(* CODESYS project genmed-LogGenTestSP14.project

Project tree, tasks and I/O mapping:
  Device : CODESYS Control for Raspberry Pi MC SL, 3S - Smart Software Solutions GmbH, version 3.5.14.20
    application Application
      libraries: Standard, * (System); VisuGlobalClientManager, * (System)
      task Task (cyclic, interval t#20ms, priority 1) calls PLC_PRG
      task DataLogHighTask (cyclic, interval t#5ms, priority 1) calls AC_CALL_DataLogHighTask_START, AC_CALL_DataLogHighTask_END
      task DataLogLowTask (cyclic, interval t#20ms, priority 10) calls AC_CALL_DataLogLowTask_START, AC_CALL_DataLogLowTask_END
      task AC_GenVisu_Task (cyclic, interval t#50ms, priority 30) calls AC_GenVisu_Prg
      task VISU_TASK (cyclic, interval 100 ms, priority 31) calls VisuElems.Visu_Prg
      program PLC_PRG [ST]
      AC_Std/
        program AC_CALL_DataLogHighTask_START [ST]
        function AC_Init [ST]
        global variables GVL_MODULE_TREE
        program AC_CALL_DataLogHighTask_END [ST]
        function AC_InitInternal [ST]
        function AC_OnlineChange [ST]
        global variables MODULE_INFOS
        program AC_CALL_DataLogLowTask_START [ST]
        program AC_CALL_DataLogLowTask_END [ST]
        global variables GVL_DataLogManager
      data type LogStruct
      data type LogUnion
      AC_Visu/
        function block AC_Visu_FB [ST]: OnFrameIndexChanged, GetModuleFrameIndex, GetAncestor
        visualisation Page_DataLogManager
        function AC_VisuInit [ST]
        visualisation Toplevel
        global variables GVL_Visu
        program AC_GenVisu_Prg [ST]
        function block AC_GlobalClientManagerListener [ST]: ClientDestroyed, ClientCreated
        global variables GVL_GlobalClientManagerListener
        function AC_RegisterVisuClientInit [ST]
      AC_FBs/
        function block AC_DataLogManager_DataLogChannel_1 [ST]
        function block AC_DataLogManager [ST]
        function block AC_DataLogManager_DataLogChannel_1_DataLogStorage_CSV [ST]
        function block AC_DataLogManager_DataLogChannel [ST]
      function block POU_Log [ST]: Prop_Log
      text DataLogConfig
    SoftMotion General Axis Pool
    I²C
    SPI
    GPIOs_A_B : GPIOs A/B, 3S - Smart Software Solutions GmbH, version 3.5.11.0
        unmapped channels: digital inputs (GPIO0..GPIO31), digital outputs (GPIO0..GPIO31)
    Onewire
    Camera device
      <Empty>
  libraries: AC_ModuleBase, * (3S - Smart Software Solutions GmbH); AC_DataLog, 3.5.14.0 (3S - Smart Software Solutions GmbH); AC_Persistence, * (3S - Smart Software Solutions GmbH); VisuSymbols, 3.5.10.0 (System)
  DataLogManager
    DataLogChannels_Role (DataLogChannels)
      DataLogChannel
        DataLogStorage_SQLite
        DataLogStorage_Role (DataLogStorage)
      DataLogChannel_1
        DataLogStorage_CSV
        A storage module. (DataLogStorage)
  AC_GENERATOR_DATA
  text list GlobalTextList
*)

// Device/Application/LogStruct
TYPE LogStruct :
STRUCT
    bNoLog : BOOL;
    {attribute 'ac_datalog'}
    bLog : BOOL;
END_STRUCT
END_TYPE

// Device/Application/LogUnion
TYPE LogUnion :
UNION
    iLog : INT;
    uiLog : UINT;
    wLog : WORD;
END_UNION
END_TYPE

// Device/Application/AC_Std/GVL_MODULE_TREE
//Code generated by Application Composer.
//Modifying generated code is not recommended!

VAR_GLOBAL
	Module_Tree: AC.ModuleTree;
	aNodes: ARRAY[0..5] OF AC.MNode;
	AC_Environment: AC.MEnv;
END_VAR

// Device/Application/AC_Std/MODULE_INFOS
//Code generated by Application Composer.
//Modifying generated code is not recommended!
{attribute 'global_init_slot' := '40000'}
{attribute 'init_on_onlchange'}

VAR_GLOBAL
	{attribute 'init_on_onlchange'}
	AC_DataLog_DataLogManager_INFO: AC.ModuleInfo := (pbyModuleType := ADR('AC_DataLog.DataLogManager'));
	{attribute 'init_on_onlchange'}
	AC_DataLog_DataLogChannel_INFO: AC.ModuleInfo := (pbyModuleType := ADR('AC_DataLog.DataLogChannel'));
	{attribute 'init_on_onlchange'}
	AC_DataLog_DataLogStorage_SQLite_INFO: AC.ModuleInfo := (pbyModuleType := ADR('AC_DataLog.DataLogStorage_SQLite'));
	{attribute 'init_on_onlchange'}
	AC_DataLog_DataLogStorage_CSV_INFO: AC.ModuleInfo := (pbyModuleType := ADR('AC_DataLog.DataLogStorage_CSV'));
END_VAR

// Device/Application/AC_Visu/GVL_Visu
//Code generated by Application Composer.
//Modifying generated code is not recommended!

VAR_GLOBAL
	g_aACVisu: ARRAY[0..7] OF AC_Visu_FB;
	AC_Visu_Dummy: AC_Visu_FB;
	g_aACVisuPtr: ARRAY[-1..127] OF POINTER TO AC_Visu_FB := [ADR(AC_Visu_Dummy), ADR(g_aACVisu[0]), ADR(g_aACVisu[1]), ADR(g_aACVisu[2]), ADR(g_aACVisu[3]), ADR(g_aACVisu[4]), ADR(g_aACVisu[5]), ADR(g_aACVisu[6]), ADR(g_aACVisu[7]), ADR(AC_Visu_Dummy), ADR(AC_Visu_Dummy), ADR(AC_Visu_Dummy), ADR(AC_Visu_Dummy), ADR(AC_Visu_Dummy), ADR(AC_Visu_Dummy), ADR(AC_Visu_Dummy), ADR(AC_Visu_Dummy), ADR(AC_Visu_Dummy), ADR(AC_Visu_Dummy), ADR(AC_Visu_Dummy), ADR(AC_Visu_Dummy), ADR(AC_Visu_Dummy), ADR(AC_Visu_Dummy), ADR(AC_Visu_Dummy), ADR(AC_Visu_Dummy), ADR(AC_Visu_Dummy), ADR(AC_Visu_Dummy), ADR(AC_Visu_Dummy), ADR(AC_Visu_Dummy), ADR(AC_Visu_Dummy), ADR(AC_Visu_Dummy), ADR(AC_Visu_Dummy), ADR(AC_Visu_Dummy), ADR(AC_Visu_Dummy), ADR(AC_Visu_Dummy), ADR(AC_Visu_Dummy), ADR(AC_Visu_Dummy), ADR(AC_Visu_Dummy), ADR(AC_Visu_Dummy), ADR(AC_Visu_Dummy), ADR(AC_Visu_Dummy), ADR(AC_Visu_Dummy), ADR(AC_Visu_Dummy), ADR(AC_Visu_Dummy), ADR(AC_Visu_Dummy), ADR(AC_Visu_Dummy), ADR(AC_Visu_Dummy), ADR(AC_Visu_Dummy), ADR(AC_Visu_Dummy), ADR(AC_Visu_Dummy), ADR(AC_Visu_Dummy), ADR(AC_Visu_Dummy), ADR(AC_Visu_Dummy), ADR(AC_Visu_Dummy), ADR(AC_Visu_Dummy), ADR(AC_Visu_Dummy), ADR(AC_Visu_Dummy), ADR(AC_Visu_Dummy), ADR(AC_Visu_Dummy), ADR(AC_Visu_Dummy), ADR(AC_Visu_Dummy), ADR(AC_Visu_Dummy), ADR(AC_Visu_Dummy), ADR(AC_Visu_Dummy), ADR(AC_Visu_Dummy), ADR(AC_Visu_Dummy), ADR(AC_Visu_Dummy), ADR(AC_Visu_Dummy), ADR(AC_Visu_Dummy), ADR(AC_Visu_Dummy), ADR(AC_Visu_Dummy), ADR(AC_Visu_Dummy), ADR(AC_Visu_Dummy), ADR(AC_Visu_Dummy), ADR(AC_Visu_Dummy), ADR(AC_Visu_Dummy), ADR(AC_Visu_Dummy), ADR(AC_Visu_Dummy), ADR(AC_Visu_Dummy), ADR(AC_Visu_Dummy), ADR(AC_Visu_Dummy), ADR(AC_Visu_Dummy), ADR(AC_Visu_Dummy), ADR(AC_Visu_Dummy), ADR(AC_Visu_Dummy), ADR(AC_Visu_Dummy), ADR(AC_Visu_Dummy), ADR(AC_Visu_Dummy), ADR(AC_Visu_Dummy), ADR(AC_Visu_Dummy), ADR(AC_Visu_Dummy), ADR(AC_Visu_Dummy), ADR(AC_Visu_Dummy), ADR(AC_Visu_Dummy), ADR(AC_Visu_Dummy), ADR(AC_Visu_Dummy), ADR(AC_Visu_Dummy), ADR(AC_Visu_Dummy), ADR(AC_Visu_Dummy), ADR(AC_Visu_Dummy), ADR(AC_Visu_Dummy), ADR(AC_Visu_Dummy), ADR(AC_Visu_Dummy), ADR(AC_Visu_Dummy), ADR(AC_Visu_Dummy), ADR(AC_Visu_Dummy), ADR(AC_Visu_Dummy), ADR(AC_Visu_Dummy), ADR(AC_Visu_Dummy), ADR(AC_Visu_Dummy), ADR(AC_Visu_Dummy), ADR(AC_Visu_Dummy), ADR(AC_Visu_Dummy), ADR(AC_Visu_Dummy), ADR(AC_Visu_Dummy), ADR(AC_Visu_Dummy), ADR(AC_Visu_Dummy), ADR(AC_Visu_Dummy), ADR(AC_Visu_Dummy), ADR(AC_Visu_Dummy), ADR(AC_Visu_Dummy), ADR(AC_Visu_Dummy), ADR(AC_Visu_Dummy), ADR(AC_Visu_Dummy), ADR(AC_Visu_Dummy), ADR(AC_Visu_Dummy), ADR(AC_Visu_Dummy), ADR(AC_Visu_Dummy), ADR(AC_Visu_Dummy)];
	g_paACVisuPtr: POINTER TO POINTER TO AC.AC_Visu_Base := ADR(g_aACVisuPtr[0]);
END_VAR

// Device/Application/AC_Std/GVL_DataLogManager
//Code generated by Application Composer.
//Modifying generated code is not recommended!

VAR_GLOBAL
	DataLogManager: AC_DataLogManager;
END_VAR

// Device/Application/AC_Visu/GVL_GlobalClientManagerListener
//Code generated by Application Composer.
//Modifying generated code is not recommended!

VAR_GLOBAL
	g_clientManagerListener: AC_GlobalClientManagerListener;
END_VAR

// Device/Application/PLC_PRG
PROGRAM PLC_PRG
VAR
    timer : Standard.TON;
    {attribute 'ac_datalog_hysteresis' := '1.745'}
    {attribute 'ac_datalog' := 'DataLogChannel'}
    iLogVar : INT;
    {attribute 'ac_datalog' := 'DataLogChannel'}
    rLogVar : REAL;
    {attribute 'ac_datalog' := 'DataLogChannel'}
    {attribute 'ac_datalog_hysteresis' := '0.745'}
    sLogVar : STRING := 'Hallo';
    //{attribute 'ac_datalog' := 'DataLogChannel'}
    arLogArray : ARRAY[0..4] OF REAL;
    
    {attribute 'ac_datalog_set_default_group' := 'DataLogChannel'}
    instStruct : LogStruct;
    
    {attribute 'ac_datalog_union_set_representant' := 'uiLog'}
    {attribute 'ac_datalog' := 'DataLogChannel_1'}
    instUnion : LogUnion;

    {attribute 'ac_datalog' := 'DataLogChannel_1'}
    {attribute 'ac_persist' := 'PersistenceChannel'}
    instFB : POU_Log;    
    
    {attribute 'ac_datalog' := 'DataLogChannel_1'}
    iLogVar2 : INT;
END_VAR

timer(IN := TRUE, PT:=T#5S);
IF timer.Q THEN
    iLogVar := iLogVar + 1;
    iLogVar2 := iLogVar;
    timer(IN := FALSE);
    rLogVar := arLogArray[2];
    instStruct.bLog := instStruct.bNoLog;
    instFB.Prop_Log := instFB.Prop_Log + 1;
END_IF

END_PROGRAM

// Device/Application/POU_Log
FUNCTION_BLOCK POU_Log
VAR_INPUT
END_VAR
VAR_OUTPUT
END_VAR
VAR
    member_1, member_2 : BOOL;
    {attribute 'ac_datalog_exclude'}
    iProp : INT;
END_VAR

{attribute 'monitoring' := 'variable'}
PROPERTY Prop_Log : INT
SET
THIS^.iProp := Prop_Log;
END_SET
GET
Prop_Log := THIS^.iProp;
END_GET
END_PROPERTY

END_FUNCTION_BLOCK

// Device/Application/AC_Std/AC_CALL_DataLogHighTask_START
//Code generated by Application Composer.
//Modifying generated code is not recommended!
PROGRAM AC_CALL_DataLogHighTask_START

//Code generated by Application Composer.
//Modifying generated code is not recommended!
DataLogManager.CallPrioHIGHStart() ;

END_PROGRAM

// Device/Application/AC_Std/AC_CALL_DataLogHighTask_END
//Code generated by Application Composer.
//Modifying generated code is not recommended!
PROGRAM AC_CALL_DataLogHighTask_END

//Code generated by Application Composer.
//Modifying generated code is not recommended!
DataLogManager.CallPrioHIGHEnd() ;

END_PROGRAM

// Device/Application/AC_Std/AC_CALL_DataLogLowTask_START
//Code generated by Application Composer.
//Modifying generated code is not recommended!
PROGRAM AC_CALL_DataLogLowTask_START

//Code generated by Application Composer.
//Modifying generated code is not recommended!
DataLogManager.CallPrioLOWStart() ;

END_PROGRAM

// Device/Application/AC_Std/AC_CALL_DataLogLowTask_END
//Code generated by Application Composer.
//Modifying generated code is not recommended!
PROGRAM AC_CALL_DataLogLowTask_END

//Code generated by Application Composer.
//Modifying generated code is not recommended!
DataLogManager.CallPrioLOWEnd() ;

END_PROGRAM

// Device/Application/AC_Visu/AC_GenVisu_Prg
//Code generated by Application Composer.
//Modifying generated code is not recommended!
PROGRAM AC_GenVisu_Prg
VAR
    i : INT ;
END_VAR

//Code generated by Application Composer.
//Modifying generated code is not recommended!
FOR i := 0 TO 7 DO
    g_aACVisu[i]() ;
END_FOR

END_PROGRAM

// Device/Application/AC_Std/AC_Init
//Code generated by Application Composer.
//Modifying generated code is not recommended!
{attribute 'linkalways'}
{attribute 'call_after_global_init_slot' := '1234'}
FUNCTION AC_Init

//Code generated by Application Composer.
//Modifying generated code is not recommended!
AC_InitInternal(FALSE);

END_FUNCTION

// Device/Application/AC_Std/AC_InitInternal
//Code generated by Application Composer.
//Modifying generated code is not recommended!
FUNCTION AC_InitInternal
VAR_INPUT
  bOnlineChange : BOOL ;
END_VAR
VAR
  hnd : AC.ModuleHandle ;
END_VAR

//Code generated by Application Composer.
//Modifying generated code is not recommended!
AC_Environment.mtree := Module_Tree ;
{IF defined(variable:AC_Environment.exts)}
	AC_Environment.exts := 0 ;
	AC_Environment.uiexts := 0 ;
{END_IF}
Module_Tree.Init(ADR(aNodes), 6);
hnd := Module_Tree.AddChild(0, DataLogManager);
DataLogManager.SetIdentification(ADR('DataLogManager'), ADR(AC_DataLog_DataLogManager_INFO), 16#2610EBE4, hnd, ADR(AC_Environment)) ;
hnd := Module_Tree.AddChild(DataLogManager, DataLogManager.INST_DataLogChannel_1);
DataLogManager.INST_DataLogChannel_1.SetIdentification(ADR('DataLogChannel_1'), ADR(AC_DataLog_DataLogChannel_INFO), 16#261012D2, hnd, ADR(AC_Environment)) ;
hnd := Module_Tree.AddChild(DataLogManager, DataLogManager.INST_DataLogChannel);
DataLogManager.INST_DataLogChannel.SetIdentification(ADR('DataLogChannel'), ADR(AC_DataLog_DataLogChannel_INFO), 16#26107E9B, hnd, ADR(AC_Environment)) ;
hnd := Module_Tree.AddChild(DataLogManager.INST_DataLogChannel_1, DataLogManager.INST_DataLogChannel_1.INST_DataLogStorage_CSV);
DataLogManager.INST_DataLogChannel_1.INST_DataLogStorage_CSV.SetIdentification(ADR('DataLogStorage_CSV'), ADR(AC_DataLog_DataLogStorage_CSV_INFO), 16#26107B70, hnd, ADR(AC_Environment)) ;
hnd := Module_Tree.AddChild(DataLogManager.INST_DataLogChannel, DataLogManager.INST_DataLogChannel.INST_DataLogStorage_SQLite);
DataLogManager.INST_DataLogChannel.INST_DataLogStorage_SQLite.SetIdentification(ADR('DataLogStorage_SQLite'), ADR(AC_DataLog_DataLogStorage_SQLite_INFO), 16#26103C5A, hnd, ADR(AC_Environment)) ;
DataLogManager.uiNumDataLogChannels := 2;
DataLogManager.AC_ARRAY_pitfDataLogChannels[0] := DataLogManager.INST_DataLogChannel;
DataLogManager.AC_ARRAY_pitfDataLogChannels[1] := DataLogManager.INST_DataLogChannel_1;
DataLogManager.pitfDataLogChannels := ADR(DataLogManager.AC_ARRAY_pitfDataLogChannels);
DataLogManager.INST_DataLogChannel.xEnable := TRUE;
DataLogManager.INST_DataLogChannel.xSaveInFirstCycle := TRUE;
DataLogManager.INST_DataLogChannel.itfDataLogStorage := DataLogManager.INST_DataLogChannel.INST_DataLogStorage_SQLite;
DataLogManager.INST_DataLogChannel_1.xEnable := TRUE;
DataLogManager.INST_DataLogChannel_1.xSaveInFirstCycle := TRUE;
DataLogManager.INST_DataLogChannel_1.itfDataLogStorage := DataLogManager.INST_DataLogChannel_1.INST_DataLogStorage_CSV;
DataLogManager.INST_DataLogChannel_1.INST_DataLogStorage_CSV.sSeperator := '||';
DataLogManager.INST_DataLogChannel_1.INST_DataLogStorage_CSV.uiBufferSize := 2000;
DataLogManager.INST_DataLogChannel_1.INST_DataLogStorage_CSV.rBufferFillLevel := 0;
DataLogManager.INST_DataLogChannel_1.INST_DataLogStorage_CSV.pbyBuffer := ADR(DataLogManager.INST_DataLogChannel_1.INST_DataLogStorage_CSV.AC_ARRAY_pbyBuffer);
IF bOnlineChange THEN
    DataLogManager.INST_DataLogChannel.tSaveCyclic := TIME#0ms;
    DataLogManager.INST_DataLogChannel_1.tSaveCyclic := TIME#0ms;
    DataLogManager.INST_DataLogChannel.INST_DataLogStorage_SQLite.sStorageName := '%CHANNEL_NAME%';
    DataLogManager.INST_DataLogChannel.INST_DataLogStorage_SQLite.uiNumMaxEntries := 0;
    DataLogManager.INST_DataLogChannel_1.INST_DataLogStorage_CSV.sStorageName := '%CHANNEL_NAME%';
END_IF
DataLogManager.Init(bOnlineChange);

END_FUNCTION

// Device/Application/AC_Std/AC_OnlineChange
//Code generated by Application Composer.
//Modifying generated code is not recommended!
{attribute 'linkalways'}
{attribute 'call_after_online_change_slot' := '1234'}
FUNCTION AC_OnlineChange

//Code generated by Application Composer.
//Modifying generated code is not recommended!
DataLogManager.OnBeforeOnlineChange();
AC_InitInternal(TRUE);
DataLogManager.OnAfterOnlineChange();

END_FUNCTION

// Device/Application/AC_FBs/AC_DataLogManager_DataLogChannel_1
//Code generated by Application Composer.
//Modifying generated code is not recommended!
FUNCTION_BLOCK AC_DataLogManager_DataLogChannel_1 EXTENDS AC_DataLog.DataLogChannel
VAR_INPUT 
    INST_DataLogStorage_CSV : AC_DataLogManager_DataLogChannel_1_DataLogStorage_CSV;
END_VAR

//Code generated by Application Composer.
//Modifying generated code is not recommended!
SUPER^();

END_FUNCTION_BLOCK

// Device/Application/AC_FBs/AC_DataLogManager_DataLogChannel_1_DataLogStorage_CSV
//Code generated by Application Composer.
//Modifying generated code is not recommended!
FUNCTION_BLOCK AC_DataLogManager_DataLogChannel_1_DataLogStorage_CSV EXTENDS AC_DataLog.DataLogStorage_CSV
VAR_INPUT 
    AC_ARRAY_pbyBuffer : ARRAY[0..1999] OF BYTE;
END_VAR

//Code generated by Application Composer.
//Modifying generated code is not recommended!
SUPER^();

END_FUNCTION_BLOCK

// Device/Application/AC_FBs/AC_DataLogManager
//Code generated by Application Composer.
//Modifying generated code is not recommended!
FUNCTION_BLOCK AC_DataLogManager EXTENDS AC_DataLog.DataLogManager
VAR_INPUT 
    INST_DataLogChannel : AC_DataLogManager_DataLogChannel;
    INST_DataLogChannel_1 : AC_DataLogManager_DataLogChannel_1;
    AC_ARRAY_pitfDataLogChannels : ARRAY[0..1] OF AC_DataLog.IDataLogChannel;
END_VAR

//Code generated by Application Composer.
//Modifying generated code is not recommended!
SUPER^();

END_FUNCTION_BLOCK

// Device/Application/AC_FBs/AC_DataLogManager_DataLogChannel
//Code generated by Application Composer.
//Modifying generated code is not recommended!
FUNCTION_BLOCK AC_DataLogManager_DataLogChannel EXTENDS AC_DataLog.DataLogChannel
VAR_INPUT 
    INST_DataLogStorage_SQLite : AC_DataLog.DataLogStorage_SQLite;
END_VAR

//Code generated by Application Composer.
//Modifying generated code is not recommended!
SUPER^();

END_FUNCTION_BLOCK

// Device/Application/AC_Visu/AC_Visu_FB
FUNCTION_BLOCK AC_Visu_FB EXTENDS AC.AC_Visu_Base
VAR_OUTPUT
    xDataLogManager : BOOL := FALSE ;
END_VAR

//Code generated by Application Composer.
//Modifying generated code is not recommended!
SUPER^();

METHOD PROTECTED OnFrameIndexChanged
VAR_INPUT
	uiIdx : UINT ;
END_VAR
CASE uiIdx OF
    0 : stAddr := AC.GetInstancePath(DataLogManager) ;
    ELSE
        stAddr := 'ERROR' ;
END_CASE
xDataLogManager := (uiIdx = 0) ;
END_METHOD

METHOD GetModuleFrameIndex : INT
VAR_INPUT
	hnd : AC.ModuleHandle ;
END_VAR
CASE hnd OF
    1 : GetModuleFrameIndex := 0 ;
    ELSE
        GetModuleFrameIndex := -1 ;
END_CASE
END_METHOD

METHOD PROTECTED GetAncestor : INT
VAR_INPUT
	uiIdx : UINT ;
END_VAR
GetAncestor := -1;
END_METHOD

END_FUNCTION_BLOCK

// Device/Application/AC_Visu/AC_VisuInit
//Code generated by Application Composer.
//Modifying generated code is not recommended!
{attribute 'linkalways'}
{attribute 'call_after_global_init_slot' := '1234'}
FUNCTION AC_VisuInit

//Code generated by Application Composer.
//Modifying generated code is not recommended!
AC_Environment.visus := g_paACVisuPtr;

END_FUNCTION

// Device/Application/AC_Visu/AC_GlobalClientManagerListener
FUNCTION_BLOCK AC_GlobalClientManagerListener IMPLEMENTS VisuGlobalClientManager.Visu_Interfaces.IGlobalClientManagerListener

//Code generated by Application Composer.
//Modifying generated code is not recommended!

METHOD ClientDestroyed
VAR_INPUT
	iGlobalClientID : INT;
	eVisuClientType : VisuGlobalClientManager.Visu_Interfaces.Visu_ClientTypeItf;
END_VAR
AC.OnClientCreatedOrDestroyed(GVL_Visu.g_aACVisuPtr[iGlobalClientID]);
END_METHOD

METHOD ClientCreated
VAR_INPUT
	iGlobalClientID : INT;
	eVisuClientType : VisuGlobalClientManager.Visu_Interfaces.Visu_ClientTypeItf;
END_VAR
AC.OnClientCreatedOrDestroyed(GVL_Visu.g_aACVisuPtr[iGlobalClientID]);
END_METHOD

END_FUNCTION_BLOCK

// Device/Application/AC_Visu/AC_RegisterVisuClientInit
//Code generated by Application Composer.
//Modifying generated code is not recommended!
{attribute 'linkalways'}
{attribute 'call_after_global_init_slot' := '1234'}
FUNCTION AC_RegisterVisuClientInit
VAR
	itfVisuGlobalClientManager2 : VisuGlobalClientManager.Visu_Interfaces.IVisuGlobalClientManager2;
END_VAR

//Code generated by Application Composer.
//Modifying generated code is not recommended!
IF __QUERYINTERFACE(VisuGlobalClientManager.Visu_Interfaces.GVL.g_GlobalClientManager, itfVisuGlobalClientManager2) THEN
	itfVisuGlobalClientManager2.AddGlobalClientManagerListener(GVL_GlobalClientManagerListener.g_clientManagerListener);
END_IF

END_FUNCTION

// Device/Application/AC_Visu/Page_DataLogManager
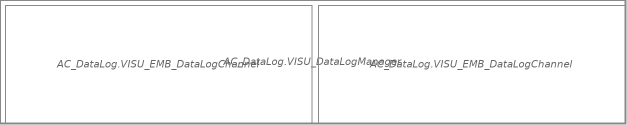
VISUALIZATION Page_DataLogManager  // 627x125
    Frame (0,0 625x123)
        shows AC_DataLog.VISU_DataLogManager(inst := DataLogManager)
    Frame (5,5 307x118)
        shows AC_DataLog.VISU_EMB_DataLogChannel(inst := DataLogManager.INST_DataLogChannel)
    Frame (318,5 307x118)
        shows AC_DataLog.VISU_EMB_DataLogChannel(inst := DataLogManager.INST_DataLogChannel_1)
END_VISUALIZATION

// Device/Application/AC_Visu/Toplevel
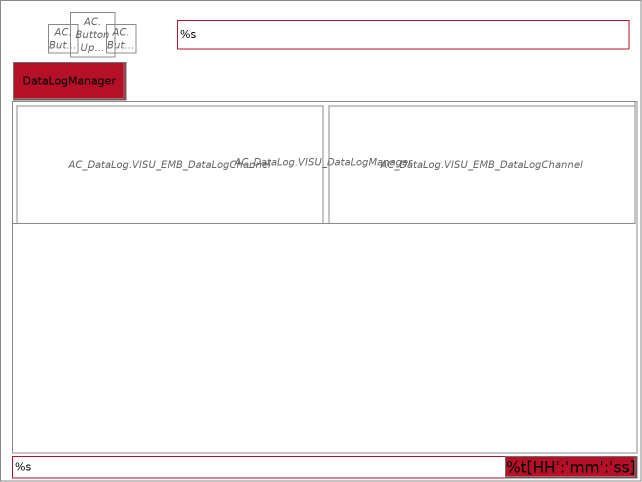
VISUALIZATION Toplevel  // 642x482
    Rectangle (10,10 630x470)
    Rectangle (10,10 630x49)
    Frame (106,24 30x29), input disabled if: g_aACVisuPtr[CURRENTCLIENTID]^.iFwdState = 2, frame switch variable: g_aACVisuPtr[CURRENTCLIENTID]^.iFwdState
        shows AC.ButtonFwd_Normal_VisuStyles()
        shows AC.ButtonFwd_MouseDown_VisuStyles()
        shows AC.ButtonFwd_Deactivated_VisuStyles()
        OnMouseDown: execute { g_aACVisuPtr[CURRENTCLIENTID]^.xFwdPressed := TRUE ; }
        OnMouseClick: execute { g_aACVisuPtr[CURRENTCLIENTID]^.xFwd := TRUE ; }
        OnMouseUp: execute { g_aACVisuPtr[CURRENTCLIENTID]^.xFwdPressed := FALSE ; }
    Frame (48,24 30x29), input disabled if: g_aACVisuPtr[CURRENTCLIENTID]^.iBackState = 2, frame switch variable: g_aACVisuPtr[CURRENTCLIENTID]^.iBackState
        shows AC.ButtonBack_Normal_VisuStyles()
        shows AC.ButtonBack_MouseDown_VisuStyles()
        shows AC.ButtonBack_Deactivated_VisuStyles()
        OnMouseDown: execute { g_aACVisuPtr[CURRENTCLIENTID]^.xBackPressed := TRUE ; }
        OnMouseClick: execute { g_aACVisuPtr[CURRENTCLIENTID]^.xBack := TRUE ; }
        OnMouseUp: execute { g_aACVisuPtr[CURRENTCLIENTID]^.xBackPressed := FALSE ; }
    Frame (70,12 45x45), input disabled if: g_aACVisuPtr[CURRENTCLIENTID]^.iUpState = 2, frame switch variable: g_aACVisuPtr[CURRENTCLIENTID]^.iUpState
        shows AC.ButtonUp_Normal_VisuStyles()
        shows AC.ButtonUp_MouseDown_VisuStyles()
        shows AC.ButtonUp_Deactivated_VisuStyles()
        OnMouseDown: execute { g_aACVisuPtr[CURRENTCLIENTID]^.xUpPressed := TRUE ; }
        OnMouseClick: execute { g_aACVisuPtr[CURRENTCLIENTID]^.xUp := TRUE ; }
        OnMouseUp: execute { g_aACVisuPtr[CURRENTCLIENTID]^.xUpPressed := FALSE ; }
    Textfield (177,20 452x29), "%s", text variable: g_aACVisuPtr[CURRENTCLIENTID]^.stAddr
    Textfield (12,456 512x22), "%s", text variable: AC.g_stVisuStatusBar
    Frame (12,101 625x352), frame switch variable: g_aACVisuPtr[CURRENTCLIENTID]^.uiCurFrameIdx
        shows Page_DataLogManager()
        shows Page_Heizung()
        shows Page_Wetter()
    Button (13,62 113x38), "DataLogManager", colour toggle: g_aACVisuPtr[CURRENTCLIENTID]^.xDataLogManager, pressed state: g_aACVisuPtr[CURRENTCLIENTID]^.xDataLogManager
        OnMouseDown: execute { g_aACVisuPtr[CURRENTCLIENTID]^.uiFrameIdx := 0 ; }
    Button (505,456 132x22), "%t[HH':'mm':'ss]", input disabled if: true
END_VISUALIZATION

(* text DataLogConfig
// DataLog configuration for for application Device.Application
// Generated automatically by GenDataLog

SEC General
  Application := Device.Application;
  ExcludedGroups := [  ];
  ToplevelInstanceNames := [ DataLogManager ];
  ToplevelFBPaths := [ GVL_DataLogManager.DataLogManager ] ;
END_SEC
SEC Channel : DataLogChannel
  Groups := [ DataLogChannel ];
  FBPath := DataLogManager.INST_DataLogChannel;
  UseHashedInstancePathesChanged := True;
END_SEC
SEC Channel : DataLogChannel_1
  Groups := [ DataLogChannel_1 ];
  FBPath := DataLogManager.INST_DataLogChannel_1;
  UseHashedInstancePathesChanged := False;
END_SEC
*)
